{attribute 'qualified_only'}
{attribute 'strict'}
{attribute 'to_string'}
TYPE E_ModuleId :
(
	GC1 := 1,
	GC2,
	LP1,
	LP2
)UDINT;
END_TYPE

(* stored: Version 1.1.0.1, ProductVersion 3.1.4026.18
   DUT E_ModuleId: Id {120572ed-5717-4c1f-b105-7b14d5843207} *)
